FUNCTION_BLOCK CalamityPumpBasic (* Basic Function Block Type *)
  (* Standard: 61499-2 *)
  (* Version 0.0, 6/26/2026, Schneider Electric, Template *)
  PACKAGE SE.Nereda;
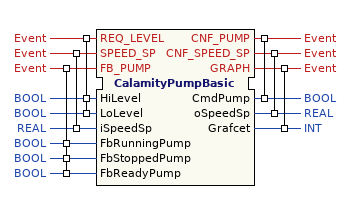
  EVENT_INPUT
    REQ_LEVEL WITH HiLevel, LoLevel; (* Normal Execution Request *)
    SPEED_SP WITH iSpeedSp;
    FB_PUMP WITH FbRunningPump, FbStoppedPump, FbReadyPump;
  END_EVENT
  EVENT_OUTPUT
    CNF_PUMP WITH CmdPump; (* Execution Confirmation *)
    CNF_SPEED_SP WITH oSpeedSp;
    GRAPH WITH Grafcet;
  END_EVENT
  VAR_INPUT
    HiLevel : BOOL;
    LoLevel : BOOL;
    iSpeedSp : REAL;
    FbRunningPump : BOOL;
    FbStoppedPump : BOOL;
    FbReadyPump : BOOL;
  END_VAR
  VAR_OUTPUT
    CmdPump : BOOL;
    oSpeedSp : REAL;
    Grafcet : INT;
  END_VAR
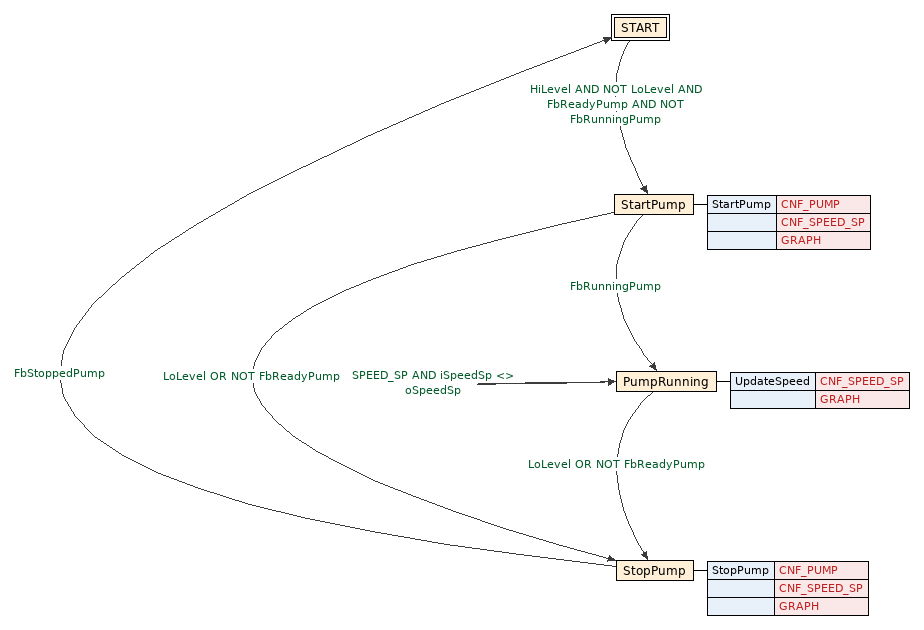
  EC_STATES
    START; (* Initial State *)
    StartPump : StartPump -> CNF_PUMP, -> CNF_SPEED_SP, -> GRAPH;
    PumpRunning : UpdateSpeed -> CNF_SPEED_SP, -> GRAPH;
    StopPump : StopPump -> CNF_PUMP, -> CNF_SPEED_SP, -> GRAPH;
  END_STATES
  EC_TRANSITIONS
    START TO StartPump := HiLevel AND NOT LoLevel AND FbReadyPump AND NOT FbRunningPump;
    StartPump TO PumpRunning := FbRunningPump;
    PumpRunning TO StopPump := LoLevel OR NOT FbReadyPump;
    StopPump TO START := FbStoppedPump;
    PumpRunning TO PumpRunning := SPEED_SP AND iSpeedSp <> oSpeedSp;
    StartPump TO StopPump := LoLevel OR NOT FbReadyPump;
  END_TRANSITIONS
  ALGORITHM StartPump IN ST:
;
CmdPump := TRUE;
oSpeedSp := iSpeedSp;
Grafcet := 1;
  END_ALGORITHM
  ALGORITHM UpdateSpeed IN ST:
;
oSpeedSp := iSpeedSp;
Grafcet := 2;
  END_ALGORITHM
  ALGORITHM StopPump IN ST:
;
CmdPump := FALSE;
oSpeedSp := 0;
Grafcet := 3;
  END_ALGORITHM
END_FUNCTION_BLOCK
